TYPE sPositionValues :
STRUCT
	q1			:LREAL;
	q2			:LREAL;
	q3			:LREAL;
	q4			:LREAL;
	q5			:LREAL;
	q6			:LREAL;
END_STRUCT
END_TYPE

(* stored: Version 1.1.0.1
   DUT sPositionValues: Id {1b5fc528-2152-4ff7-b7cb-3d89b85a7d5f} *)
